{attribute addProperty BoxType "EPP1816-3008-0016"}
{attribute addProperty Id "ErrorBIT10.1257TxPDO_ToggleBIT10.12516"}
{attribute addProperty CRC "2662626009"}
{attribute addProperty SizeInBites "16"}
{attribute addProperty SizeInBytes "2"}
TYPE Status_9EB472D9 :
STRUCT
	{attribute 'hide'}
	reserve_1_BIT_0 : BIT;
	{attribute 'hide'}
	reserve_1_BIT_1 : BIT;
	{attribute 'hide'}
	reserve_1_BIT_2 : BIT;
	{attribute 'hide'}
	reserve_1_BIT_3 : BIT;
	{attribute 'hide'}
	reserve_1_BIT_4 : BIT;
	{attribute 'hide'}
	reserve_1_BIT_5 : BIT;
	{attribute addProperty Name "Error"}
	Error : BIT;
	{attribute 'hide'}
	reserve_2 : BYTE;
	{attribute addProperty Name "TxPDO_Toggle"}
	TxPDO_Toggle : BIT;
END_STRUCT
END_TYPE

(* stored: Version 1.2.0.0, ProductVersion 3.1.4024.9
   DUT Status_9EB472D9: Id {dc0f22bb-69c4-4918-8bcd-e363d970941c} *)
